PROGRAM main
VAR
	Waktu_Blink : time := T#1s;
	Timer1 : TON;
	Timer2 : TON;
	LED_out AT %QX0.0 : bool;
	WIFI_SCANNER1 : Wifi_Scanner;
END_VAR

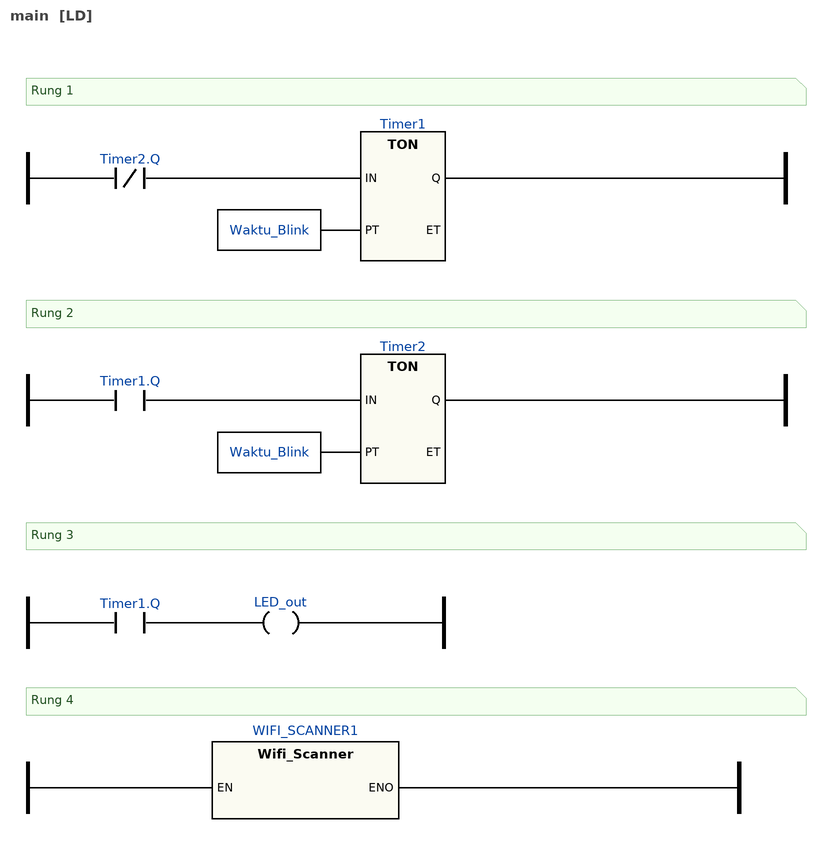
(* LD diagram, written out as Structured Text *)
(* Rung 1 *)
(* Rung 2 *)
(* Rung 3 *)
LED_out := Timer1.Q;
Timer1(IN := NOT Timer2.Q, PT := Waktu_Blink);
Timer2(IN := Timer1.Q, PT := Waktu_Blink);
(* Rung 4 *)
WIFI_SCANNER1();
END_PROGRAM
